// TIA Portal V17 export
// export: Created 2025-08-05T09:35:58.8277614Z, ExportSetting WithDefaults, DisplayName Totally Integrated Automation Portal, DisplayVersion V17, DisplayName TIA Portal Openness, DisplayVersion V17, DisplayName TIA Portal Version Control Interface, DisplayVersion V17, DisplayName SINAMICS Startdrive Advanced, DisplayVersion V17, DisplayName SINAMICS Startdrive G130, G150, S120, S150, SINAMICS MV, S210, DisplayVersion V17, DisplayName SINAMICS Startdrive G110M, G120, G120C, G120D, G120P, G115D, DisplayVersion V17, DisplayName STEP 7 Professional, DisplayVersion V17, DisplayName STEP 7 Safety, DisplayVersion V17, DisplayName WinCC Advanced, DisplayVersion V17
DATA_BLOCK "Control_DB"   // DB2
VERSION : 0.1
// stored: AutoNumber true, DBAccessibleFromOPCUA true, DBAccessibleFromWebserver true, InstanceOfName Control, InstanceOfType FB
"Control"
   // VAR_INPUT
   //    iGraph_Step_1 : Bool;
   //    iInstance_Index : DInt;
   // END_VAR
   // VAR_IN_OUT
   //    ioGraph_Job_Select : Int;
   // END_VAR
   // VAR
   //    sStep : DInt;
   //    sNo_Faults_Active : Bool;
   //    Step_Delay { S7_SetPoint := 'True'} : TON_TIME;
   //    sCounter_Done : Bool;
   //    sCTU : IEC_COUNTER;
   //    sWeldJob { S7_SetPoint := 'True'} : Byte;
   //    sDelayDone : Bool;
   // END_VAR
BEGIN
END_DATA_BLOCK
